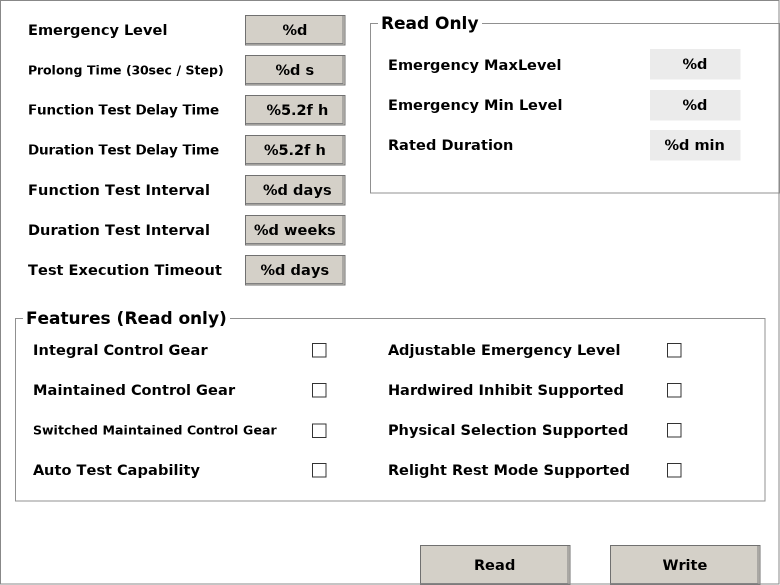
VISUALIZATION Visu_Part202Parameters  // 780x585
    Button (610,545 150x40), "Write"
        OnMouseClick: execute { DALI_Commissioning.fbPart202Emergency.bWrite:=TRUE; }
    GroupBox (15,310 750x191), "Features (Read only)"
        Textfield (15,25 250x30), "Integral Control Gear"
        Textfield (15,65 250x30), "Maintained Control Gear"
        Checkbox (295,105 30x31), variable: DALI_Commissioning.fbPart202Emergency.bSwitchtedMaintainedControlGear, input disabled if: TRUE
        Checkbox (295,25 30x30), variable: DALI_Commissioning.fbPart202Emergency.bIntegralControlGear, input disabled if: TRUE
        Checkbox (295,65 30x30), variable: DALI_Commissioning.fbPart202Emergency.bMaintainedControlGear, input disabled if: TRUE
        Textfield (370,105 250x30), "Physical Selection Supported"
        Textfield (15,145 250x30), "Auto Test Capability"
        Textfield (370,25 250x30), "Adjustable Emergency Level"
        Textfield (370,65 250x30), "Hardwired Inhibit Supported"
        Textfield (370,145 250x30), "Relight Rest Mode Supported"
        Checkbox (650,25 30x30), variable: DALI_Commissioning.fbPart202Emergency.bAdjustableEmergencyLevel, input disabled if: TRUE
        Checkbox (650,65 30x30), variable: DALI_Commissioning.fbPart202Emergency.bHardwiredInhibitSupported, input disabled if: TRUE
        Checkbox (650,105 30x30), variable: DALI_Commissioning.fbPart202Emergency.bPhysicalSelectionSupported, input disabled if: TRUE
        Checkbox (650,145 30x30), variable: DALI_Commissioning.fbPart202Emergency.bRelightinRestModeSupported, input disabled if: TRUE
        Textfield (15,105 250x30), "Switched Maintained Control Gear"
        Checkbox (295,145 30x30), variable: DALI_Commissioning.fbPart202Emergency.bAutoTestCapability, input disabled if: TRUE
    Textfield (25,15 200x30), "Emergency Level"
    Textfield (25,95 200x30), "Function Test Delay Time"
    Textfield (25,135 200x30), "Duration Test Delay Time"
    Button (245,15 100x30), "%d", text variable: DALI_Commissioning.fbPart202Emergency.nEmergencyLevel
        OnMouseClick: write the text variable via Default, min 0, max 255, title "Emergency Level"
    Button (245,95 100x30), "%5.2f h", text variable: DALI_Commissioning.fbPart205Incandescent.fLoadRating
        OnMouseClick: write the text variable via Default, min 0, max 16384, title "Function Test Delay Time"
    Button (245,135 100x30), "%5.2f h", text variable: DALI_Commissioning.fbPart202Emergency.fDurationTestDelayTimeVisu
        OnMouseClick: write the text variable via Default, min 0, max 16384, title "Duration Test Delay Time"
    Textfield (25,55 200x30), "Prolong Time (30sec / Step)"
    Button (245,55 100x30), "%d s", text variable: DALI_Commissioning.fbPart202Emergency.nProlongTime
        OnMouseClick: write the text variable via Default, min 0, max 255, title "Prolong Time"
    Textfield (25,255 200x30), "Test Execution Timeout"
    Button (245,255 100x30), "%d days", text variable: DALI_Commissioning.fbPart202Emergency.nTestExecutionTimeout
        OnMouseClick: write the text variable via Default, min 0, max 255, title "Test Execution Timeout"
    GroupBox (370,15 410x178), "Read Only"
        Textfield (15,115 220x30), "Rated Duration"
        Textfield (15,75 220x30), "Emergency Min Level"
        Textfield (15,35 220x30), "Emergency MaxLevel"
        Textfield (280,34 90x30), "%d", text variable: DALI_Commissioning.fbPart202Emergency.nEmergencyMaxLevel
        Textfield (280,75 90x30), "%d", text variable: DALI_Commissioning.fbPart202Emergency.nEmergencyMinLevel
        Textfield (280,115 90x30), "%d min", text variable: DALI_Commissioning.fbPart202Emergency.nRatedDuration
    Textfield (25,175 200x30), "Function Test Interval"
    Textfield (25,215 200x30), "Duration Test Interval"
    Button (245,175 100x30), "%d days", text variable: DALI_Commissioning.fbPart202Emergency.nFunctionTestInterval
        OnMouseClick: write the text variable via Default, min 0, max 255, title "Function Test Delay Time"
    Button (245,215 100x30), "%d weeks", text variable: DALI_Commissioning.fbPart202Emergency.nDurationTestInterval
        OnMouseClick: write the text variable via Default, min 0, max 255, title "Duration Test Delay Time"
    Button (420,545 150x40), "Read"
        OnMouseClick: execute { DALI_Commissioning.fbPart202Emergency.bReadParameter:=TRUE; }
END_VISUALIZATION

(* stored: Version 1.1.0.1
   Visu Visu_Part202Parameters: Id {69cd5b41-b20b-4093-9d10-51d44b3ad955} *)
